# B&R Automation Studio project ACOPOSInverterTool
Automation Studio 4.12.3.127 SP; technology packages: mapp 5.23.0, mappFramework 1.0.0, mappMotion 5.23.0, mappView 5.23.0

## Configuration Config1

CPU 4PPC70.0573-20B, AutomationRuntime E4.93, Build 4.1.2, Safety 0.0, Vc V4.72.5

### Task classes (Cpu.sw)
```
Cyclic#4:
  Main <- Main.prg
NcDataObjects: mcdrivelog
Binaries: TCLang, arsvcreg, FWRules, mvLoader, TCData, udbdef, arflatprv, arcoal, iomap, asfw, Role, ashwd, Config, Config_1, TC, arconfig, sysconf, User, ashwac
Libraries: AsEPL, runtime, MpServer, MpAlarmX, MpBase, astime, MpRecipe, sys_lib, MpCom, AsIecCon, AsMath, asstring, FileIO, AsXml, standard, ArEventLog, McBase, arssl, SfDomVis, MpSfDomMgr, dataobj, asiodiag, SfDomDrv, aruser, asusb, AsTCP, MpAxis, McAxis, McAcpAx, AsIORTI
```

### Hardware
```
4PPC70_0573_20B : 4PPC70.0573-20B v1.5.4.0
  Connector IF2:
    ActivateDevice = 1
    Mode = Manual
    InternetAddress = 192.168.0.20
    SubnetMask = 255.255.255.0
    InaPort = 11160
    ActivateSnmp = 2
    ActivateModbus = 1
    NumSlaves = -1
    NumAllBlocks = -1
    MemSizeIn = -1
    MemSizeOut = -1
    ModbusSlaveGrey = 1
  ConfigurationID = ACOPOSInverterTool_Config1
  Simulation = 1
  XLinkUseDefault = 0
  XLinkDuration = 2000
  Cyclic1Duration = 2000
  Cyclic1Tolerance = 0
  FileDevice1
  FileDeviceName1 = USER
  FileDevicePath1 = USER_PATH
  ActivateOpcUa = 1
  OpcUaInformationModels_PV_Version = 1
  KeyMappingFile = VC\4PPC70_0573_20B.dis
8I66xxxxxxx.0P-xxx : 8I66xxxxxxx.0P-xxx v2.5.1.0  [PLK1 -> 4PPC70_0573_20B.IF1 (NodeNumber=2) [Cable Type=PowerlinkCable, Length=10, Version=1.0.0.3]]
  Supervision = off
  FunctionModel = Standard
  UnitOfSetpoint = Rpm
  IOM_AIDP1 = RFR_D
  IOM_AIDP2 = FRO_D
  IOM_AIDP3 = OTRN
  IOM_AIDP4 = UOP
  IOM_AIDP5 = LCR
  IOM_AIDP6 = SLCR
  IOM_AIDP7 = OPR
  IOM_AIDP8 = ULN
  IOM_AIDP9 = THR
  IOM_AIDP10 = THD
  FunctionModel_ACPi = Template50_SYN
  Sel_NameplateMask = 8Ix6T200037_IEC
  Sel_TUN = MANU
  Sel_References = Hz
  Cfg_FLR = 1
```

### IoMap.iom - 4PPC70_0573_20B/IoMap.iom
```iecst
VAR_CONFIG
	::Main:controlWord AT %QW."8I66xxxxxxx.0P-xxx".CMDD_Output;
	::Main:errorWord AT %IW."8I66xxxxxxx.0P-xxx".ERRD_Input;
	::Main:statusWord AT %IW."8I66xxxxxxx.0P-xxx".ETAD_Input;
	::Main:hmiCom.cmd.Speed AT %QW."8I66xxxxxxx.0P-xxx".LFRD_Output;
	::Main:hmiCom.cmd.ActualSpeed  AT %IW."8I66xxxxxxx.0P-xxx".RFRD_Input;
	::Main:hmiCom.cmd.Freq AT %IW."8I66xxxxxxx.0P-xxx".FRO_Input;
	::Main:hmiCom.cmd.ActualFreq AT %IW."8I66xxxxxxx.0P-xxx".RFR_Input;
END_VAR
```

## Logical view

Binary libraries used (declarations not repeated): operator, runtime, astime, AsIecCon, AsEPL, sys_lib, AsMath, asstring, FileIO, AsXml, standard, ArEventLog, AsTCP, McBase, MpAxis, McAcpAx, McAxis, MpBase, MpRecipe, MpAlarmX, MpCom 5.23.0, MpServer, AsIORTI


### Program Logical/Main (IEC)

#### Main.st - Init, cyclic, exit code
```iecst
//
PROGRAM _INIT
//
//	(*Enable FB Blocks*) // ???
//	eplWriteBlock.enable 	:= TRUE;
//	eplReadBlock.enable 	:= TRUE;
//
END_PROGRAM
//
PROGRAM _CYCLIC
//
//	//Mappview String Handling Task
	stringhandling;
//
//	//By Default Remove Ability to Control Axis
//	//controlEnable := FALSE;
//
//	//Assign pDevice
//
//	IF hmiCom.PowerLinkPathDefault THEN
//		//If a null pointer is specified, the function block uses the first POWERLINK interface
//		eplReadBlock.pDevice 	:= 0;
//		eplWriteBlock.pDevice 	:= 0;
//	ELSIF NOT hmiCom.PowerLinkPathDefault THEN
//
//		pDevice :=
//		eplReadBlock.pDevice 	:= ADR(pDevice);
//		eplWriteBlock.pDevice 	:= ADR(pDevice);
	//Assign NodeNumber from Vis
	eplReadBlock.node		:= hmiCom.NodeNumber;
	eplWriteBlock.node		:= hmiCom.NodeNumber;
//
//
	CASE state OF

		WAIT:

			//Run Startup Routine
			IF startupRoutine AND hmiCom.NodeNumber <> 0 THEN
				startup;
			END_IF

			//Run Main Routine
			IF startupDone THEN
				j := 0;
				i := 0;
				startupRoutine := FALSE;
				state := RUN;
			END_IF

		RUN:

			CASE runstate OF

				WAITING:

					hmiCom.Reading := FALSE;
					hmiCom.Writing := FALSE;

					IF hmiCom.cmd.loadParams = 1 THEN
						hmiCom.status.readInpr := TRUE;
						hmiCom.status.ReadDone := FALSE;
						runstate := READING;
					END_IF

					IF hmiCom.cmd.saveParams = 1 THEN
						hmiCom.status.writeInpr := TRUE;
						hmiCom.status.WriteDone := FALSE;
						runstate := WRITING;
					END_IF

				READING:
					hmiCom.Reading := TRUE;
					CASE readstate OF
						READPARAMS:
							IF readBools[i] THEN 		// readBools[i] should all be 1. Added for future use
								eplReadBlock.enable			:= TRUE;
								eplReadBlock.index 			:= eplReadBuffer[i].index;
								eplReadBlock.subindex 		:= eplReadBuffer[i].subindex;
								eplReadBlock.datalen 		:= 2;	//2 bytes
								eplReadBlock.pData 		:= eplReadBuffer[i].pData;
								eplReadBuffer[i].status 	:= eplReadBlock.status;
								eplReadBuffer[i].errorinfo	:= eplReadBlock.errorinfo;
							END_IF

							//Check For Error, then move to iterate counter
							IF eplReadBlock.status = 0 THEN
								readstate 					:= ITERATEREADCOUNT;
							ELSIF NOT (eplReadBlock.status = 0 OR eplReadBlock.status = 65535 OR eplReadBlock.status = 65534) THEN
								readstate := READERROR;
								state := GLOBALERROR;
							END_IF

						ITERATEREADCOUNT:

							//Turn off enable
							eplReadBlock.enable	:= FALSE;

							//Iterate Counter
							IF i = MAXINDEX THEN
//								hmiCom.status.readInpr := FALSE;
//								hmiCom.status.ReadDone := TRUE;
								i := 0;
								readstate := READPARAMS;
								runstate := WAITING;
								hmiCom.status.readInpr := FALSE;
								hmiCom.status.ReadDone := TRUE;
							ELSE
								i := i + 1;
							END_IF
							//Send Back to Reading State
							readstate 	:= READPARAMS;

						READERROR:

							IF hmiCom.cmd.Reset = TRUE THEN

							END_IF

					END_CASE

				WRITING:
					hmiCom.Writing := FALSE;
					CASE writestate OF

						WRITEPARAMS:

							IF writeBools[j] THEN
								eplWriteBlock.index				:= eplReadBuffer[j].index;
								eplWriteBlock.subindex			:= eplReadBuffer[j].subindex;
								eplWriteBlock.datalen 			:= SIZEOF(readData.ADC);	//Any will do since the max is 2 bytes
								eplWriteBlock.pData 			:= eplReadBuffer[i].pData;
								eplWriteBuffer[j].status 		:= eplWriteBlock.status;
								eplWriteBuffer[j].errorinfo		:= eplWriteBlock.errorinfo;

								eplReadBlock.enable			:= TRUE;
							END_IF

							IF eplWriteBlock.status = 65535 THEN
								writestate 					:= ITERATEWRITECOUNT;
							END_IF

						ITERATEWRITECOUNT:
							//Turn off enable
							eplWriteBlock.enable	:= FALSE;

							//Iterate Counter
							IF j = MAXINDEX THEN
								j := 0;
								hmiCom.status.writeInpr := FALSE;
								hmiCom.status.WriteDone := TRUE;
								writestate := WRITEPARAMS;
								runstate := WAITING;
							ELSE
								j := j + 1;
							END_IF

							//Send Back to writing state
							writestate 	:= WRITEPARAMS;

						WRITEERROR:

					END_CASE

			END_CASE

		GLOBALERROR:

	END_CASE
//
//
//
	eplWriteBlock();

IF startupDone THEN
	eplReadBlock();
END_IF

END_PROGRAM
//
PROGRAM _EXIT
//	(* Insert code here *)
//
END_PROGRAM
//
```

#### Types.typ - Local data types
```iecst
(**********************************HMI VARIABLES***********************************************************)

TYPE
	hmiCommTyp : 	STRUCT  (*HMI communication structure*)
		ReadWriteBuffer : DataBufferTyp; (*Command to write*)
		InverterModel : invertermodel_enum;
		InverterModelInt : USINT;
		InverterModelString : STRING[20];
		MotorType : motortype_enum;
		PowerLinkPathDefault : BOOL; (*Set to true if there's only 1 powerlink interface on the PC*)
		PowerLinkPath : powerlinkPathTyp;
		NodeNumber : USINT; (*Node number of ACOPOS Inverter*)
		Params : paramsTyp; (*Data used in ParamsContent*)
		cmd : hmiCmdTyp;
		status : hmiStatusTyp;
		unitMonitoring : unitMonitoringTyp;
		Writing : BOOL;
		Reading : BOOL;
		selectedNRDIndex : USINT;
		selectedSFTValue : STRING[3];
		selectedSTFInt : USINT;
		selectedCFTValue : STRING[3];
		selectedCFTInt : USINT;
		selectedCTTValue : STRING[3];
		selectedCTTint : USINT;
		selectedAstValue : STRING[3];
		selectedInverter : STRING[80];
		selectedInverterINT : USINT;
		selectedMotorType : STRING[3];
		selectedMotorINT : USINT;
	END_STRUCT;
	invertermodel_enum :
		( (*ACOPOS Inverter Model enumeration*)
		P66 := 66,
		P76 := 76,
		P86 := 86
		);
	motortype_enum :
		(
		Asynchronous := 0,
		Synchronous := 1
		);
	powerlinkPathTyp : 	STRUCT  (*Carries path strings to build "SL<x>.SS<y>.IF<Z>"*)
		SLnumber : STRING[8]; (*SLx*)
		SSnumber : STRING[8]; (*SSy*)
		IFnumber : STRING[8]; (*IFz*)
	END_STRUCT;
	hmiCmdTyp : 	STRUCT
		Speed : INT;
		ActualSpeed : INT;
		Freq : INT;
		ActualFreq : INT;
		CMDD : UINT;
		loadParams : BOOL;
		saveParams : BOOL;
		Reset : BOOL;
	END_STRUCT;
	hmiStatusTyp : 	STRUCT
		ERRD : STRING[20];
		ETAD : STRING[20];
		FirmwareVersion : STRING[20];
		readInpr : BOOL;
		writeInpr : BOOL;
		ReadDone : USINT;
		WriteDone : USINT;
	END_STRUCT;
END_TYPE

(**********************************State Enumerations*********************************************************)

TYPE
	state_enum :
		(
		WAIT,
		RUN,
		GLOBALERROR
		);
	runstate_enum :
		(
		WAITING,
		READING,
		WRITING
		);
	startupstate_enum :
		(
		INITIALIZE,
		COPY,
		FIRSTREAD,
		DONE
		);
	readstate_enum :
		(
		READPARAMS,
		ITERATEREADCOUNT,
		READERROR
		);
	writestate_enum :
		(
		WRITEPARAMS,
		ITERATEWRITECOUNT,
		WRITEERROR,
		ALGR (*Status word of user defined alarm groups*)
		);
END_TYPE

(**********************************Parameter Structures******************************************************)

TYPE
	eplParTyp : 	STRUCT
		index : UINT; (*Number of the index entry to be written.
*)
		subindex : USINT; (*Number of the subindex entry to be written.
*)
		pData : UDINT; (*Pointer to the data to be written. This data must remain constant as long as the function block returns ERR_BUSY.
*)
		datalen : UDINT; (*Length of the data to be written.
*)
		status : UINT; (*Error number (0 = no error).
*)
		errorinfo : UDINT; (*SDO Abort Code (if status = ERR_ASEPL_ACCESS_FAILED)
*)
		name : STRING[50]; (*Name of Parameter*)
		measurementUnit : measurementunit_enum; (*Unit of measurement for the data*)
		conversionFactor : REAL; (*Conversion factor from data to measurement unit*)
	END_STRUCT;
	DataBufferTyp : 	STRUCT
		NSP : UINT;
		FRS : UINT;
		UNS : UINT;
		NCR : UINT;
		COSINE : UINT;
		NPR : UINT;
		TUN : WORD; (*0 - no action, 1- tune, 2 - delete tuning*)
		RSA : UINT;
		LFA : UINT;
		IDA : UINT;
		TRA : UINT;
		SFR : UINT;
		SFT : WORD; (*Heat Optimized (1), Noise Optimized (2)*)
		NRD : USINT; (*Vary PWM period for Noise reduction- No (0), Yes (1)*)
		CTT : WORD; (*(UUC)/Sensorless Flux Vector 	(0)
							 (STD)/Standard 			  	(3)
							 (UF5)/ (V/F 5pts) 				(4)
							 (SYN)/ Synchronous motor		(5)
							 (UFQ)/ (V/F QUAD.) 			(6)
							 (NLD)/Energy Saving			(7)*)
		SPGU : UINT; (*For Standard mode: *)
		SPG : UINT; (*For Vector control:*)
		FFH : UINT;
		CRTF : UINT;
		SLP : UINT;
		UFR : UINT;
		BOA : WORD; (*Boost Enum, 0 Boost inactive, 1 boost dynamic, 2 boost static*)
		FAB : UINT;
		BOO : INT;
		PFL : UINT;
		F1 : UINT;
		U1 : UINT;
		F2 : UINT;
		U2 : UINT;
		F3 : UINT;
		U3 : UINT;
		F4 : UINT;
		U4 : UINT;
		F5 : UINT;
		U5 : UINT;
		SIT : UINT;
		SFC : UINT;
		JFH : UINT;
		JPF : UINT;
		JF2 : UINT;
		JF3 : UINT;
		SPA : UINT;
		SPAT : UINT;
		SPD : UINT;
		SPDT : UINT;
		RPT : WORD; (*Enum - Linear Ramp (0), S-ramp (1), U-Ramp (2), Customized (3)*)
		ADC : WORD; (*Enum - No DC inject(0), Yes (1), Continuous DC inj brake (2)*)
		FLR : WORD; (*Enum - catch spinning loads No(0), yes(1)*)
		SDC1 : UINT;
		TDC1 : UINT;
		SDC2 : UINT;
		TDC2 : UINT;
		BRA : WORD; (*Enum - Braking cmd transistor(No) (0), Dec ramp adapt assinged (YES) (1), Dynamic high torque (2)*)
		DCF : UINT;
		IDC : UINT;
		TDI : USINT;
		IDC2 : UINT;
		TDC : UINT;
		ULT : UINT;
		LUL : UINT;
		RMUD : UINT;
		LUN : UINT;
		FTU : UINT;
		TOL : UINT;
		LOC : UINT;
		FTO : UINT;
		ITH : UINT;
		I2TA : UINT; (*Enumeration - 0 (no), 1 (yes)*)
		OTR : USINT; (*Monitored Value for Torque*)
		MAINS : UINT;
		PPNS : UINT; (*Synchronous Motor Pole Pair*)
		NSPS : UINT; (*Sync motor speed*)
		NCRS : UINT; (*Sync motor current*)
		TQS : UINT; (*Sync motor torque*)
		RSAS : UINT; (*Stator resistance (Sync)*)
		LDS : UINT; (*Direct inductance (Sync)*)
		LQS : UINT; (*Quadrature Inductance (Sync)*)
		PHS : UINT; (*Sync EMF (Voltage) constant*)
		AST : UINT; (*Synchronous Motor Construction Type*)
	END_STRUCT;
	paramsTyp : 	STRUCT
		UnitMonitoring : unitMonitoringTyp; (*Datapoints used in Units/Monitoring tab*)
	END_STRUCT;
	unitMonitoringTyp : 	STRUCT
		MeasurementUnit : measurementunit_enum;
		Units : ARRAY[0..7]OF unitTyp;
	END_STRUCT;
	unitTyp : 	STRUCT
		Unit : unit_enum; (*Unit being monitored*)
		String : STRING[80]; (*String of Description*)
		PowerlinkIndex : UINT; (*Powerlink Index*)
		PowerlinkSubindex : UINT; (*Powerlink Subindex*)
	END_STRUCT;
	measurementunit_enum :
		(
		Undefined := 0,
		Hz := 1, (*Hertz*)
		RPM := 2, (*RPM*)
		Volts := 3, (*Volts*)
		Amps := 4, (*Amperes*)
		Percent := 5, (*%*)
		NewtonMeter := 6, (*Newton-Meter*)
		Seconds := 7, (*Seconds*)
		Ohm := 8, (*Ohm*)
		Millihenry := 9 (*mH*)
		);
	unit_enum :
		( (*Enumeration containing the units that can be monitored on the inverter*)
		UNDEFINED, (*undefined*)
		HMIS, (*Device specific error code*)
		ETI, (*Internal status word*)
		THR, (*Thermal status of motor (i^2 * t)*)
		THD, (*Thermal status of drive [%]*)
		I2TM, (*Overcurrent status of motor (I^2 * t)[%]*)
		PTCI, (*Status word of PTC on DI6*)
		ALGROUP, (*Status word of user defined alarm groups*)
		STOS, (*Status word of STO (safe torque off)*)
		SS1S, (*Status word of SS1 (safe speed 1)*)
		SLSS, (*Status word of SLS (safely limit speed)*)
		SMSS, (*Status word of SMS (safe maximum speed)*)
		GDLS, (*Status word of GDL (guard door locking)*)
		ETAD, (*Status word (as BOOL)*)
		RFR, (*Frequency value [Hz] (PWM output)*)
		SRFR, (*unfiltered raw value of RFR [Hz]*)
		FRO, (*Frequency reference after a ramp [Hz] (value for PWM control)*)
		FRH, (*Frequency reference after n limitation [Hz] (value before ramp)*)
		FRHD, (*Speed reference after n limitation [rpm]*)
		OTR, (*Torque [%] (according to DS402)*)
		SOTR, (*unfiltered incremental value of OTR*)
		OTRN, (*Torque [Nm]*)
		UOP, (*Voltage [V] (PWM output) *)
		LCR, (*Current [A] (PWM output)*)
		SLCR, (*unfiltered raw value of LCR [A]*)
		OPR, (*Power [%] (PWM output)*)
		SOPR, (*unfiltered raw value of OPR [%]*)
		ULN, (*Mains voltage level [V]*)
		SULN, (*unfiltered raw valueof ULN [V]*)
		AI1R, (*Status word of analog input 1*)
		AI1RUINT, (*Status word (as UINT)*)
		AI2R, (*Status word of analog input 2*)
		AI2RUINT, (*Status word (as UINT)*)
		AI3R, (*Status word of analog input 3*)
		AI3RUINT, (*Status word (as UINT)*)
		IL1R, (*Status word of digital inputs*)
		IL1RBOOL, (*Status word (as BOOL)*)
		HSC, (*Edge counter on DI5*)
		PIFR, (*Pulse input on DI5 [0 .. 8192]*)
		PFRC, (*Pulse input on DI5 [Hz] *)
		FQS, (*Frequency meter on DI5 [Hz] (processed value)*)
		AO1I, (*Status word of analog output 1*)
		OL1I, (*Status word of digital outputs*)
		OL1IBOOL, (*Status word (as BOOL)*)
		NCRS (*Set to NCR(S) (motor nominal current)*)
		);
	ast_change_enum :
		(
		NOCHANGE,
		VISCHANGE,
		DRIVECHANGE
		);
END_TYPE

(***********************************Parameter enumerations************************************************)
```

#### Variables.var - Local variables
```iecst
(*************************************EPL Stuff************************************************************************)
VAR
	eplWriteBlock : EplSDOWrite; (*This function block is used to write a node's object entries when using an SDO transfer that is constantly running in the background.
*)
	eplReadBlock : EplSDORead; (*This function block is used to read a node's object entries when using an SDO transfer that is constantly running in the background.
*)
	eplReadBuffer : ARRAY[0..MAXINDEX] OF eplParTyp; (*Array of Inputs for the Read FB*)
	eplWriteBuffer : ARRAY[0..MAXINDEX] OF eplParTyp; (*Array of Inputs for the Write FB (Open to see parameters)*)
	readBools : ARRAY[0..MAXINDEX] OF BOOL;
	writeBools : ARRAY[0..MAXINDEX] OF BOOL;
	readData : DataBufferTyp;
	writeData : DataBufferTyp;
	pDevice : STRING[80]; (*Device name of the POWERLINK interface (syntax: SL<x>.SS<y>.IF<z>). If a null pointer is specified, the function block uses the first POWERLINK interface on the system.
*)
	state : state_enum; (*State enumeration variable*)
	runstate : runstate_enum;
	readstate : readstate_enum; (*State enumeration variable*)
	writestate : writestate_enum; (*State enumeration variable*)
	startupstate : startupstate_enum;
	aststate : ast_change_enum;
	i : USINT; (*for loop variable*)
	j : USINT; (*loop variable 2*)
	k : USINT; (*loop variable 3*)
END_VAR
VAR CONSTANT
	MAXINDEX : USINT := 77; (*Maximum index*)
END_VAR
VAR
	hmiCom : hmiCommTyp;
	addressBook : USINT;
	startupRoutine : BOOL;
	startupDone : BOOL;
	oldAstVis : STRING[3];
	oldAstDrive : UINT;
END_VAR
(**************************************Test Stuff***********************************************************************)
VAR
	controlWord : UINT; (*CMDD*)
	errorWord : UINT; (*ERRD*)
	statusWord : UINT; (*ETAD*)
	setpointRead : INT; (*FROD*)
	setpointWrite : INT; (*LFRD*)
	feedbackValue : INT; (*RFRD*)
	controlEnable : BOOL; (*Boolean to prevent writing to EPL while controlling the axis*)
	firmwareVersion : UDINT;
	hardwareVariant : UDINT;
END_VAR
(*************************************Hmi Comm Stuff********************************************************************)
VAR
	comm : hmiCommTyp;
END_VAR
```

#### stringhandling.st
```iecst
ACTION stringhandling:

		//Inverter Model

		//Motor Type

		hmiCom.selectedMotorINT := STRING_TO_USINT(hmiCom.selectedMotorType);

		//Monitored Units

		FOR k := 0  TO 7 DO
			CASE hmiCom.Params.UnitMonitoring.Units[i].Unit OF

			UNDEFINED:
				hmiCom.Params.UnitMonitoring.Units[k].String 			:= 'Undefined';
				hmiCom.Params.UnitMonitoring.Units[k].PowerlinkIndex 	:= 16#0;
				hmiCom.Params.UnitMonitoring.Units[k].PowerlinkSubindex := 16#0;
				hmiCom.Params.UnitMonitoring.MeasurementUnit 			:= Undefined;
			HMIS:
				//A bunch of different HMIS in the sheet, using the first
				hmiCom.Params.UnitMonitoring.Units[k].String 			:= 'Device specific error code';
				hmiCom.Params.UnitMonitoring.Units[k].PowerlinkIndex 	:= 16#202B;
				hmiCom.Params.UnitMonitoring.Units[k].PowerlinkSubindex := 16#16;
				hmiCom.Params.UnitMonitoring.MeasurementUnit 			:= Undefined;
			ETI:
				//A bunch of different ETI in the sheet, using the first
				hmiCom.Params.UnitMonitoring.Units[k].String 			:= 'Internal status word';
				hmiCom.Params.UnitMonitoring.Units[k].PowerlinkIndex 	:= 16#202A;
				hmiCom.Params.UnitMonitoring.Units[k].PowerlinkSubindex := 16#15;
				hmiCom.Params.UnitMonitoring.MeasurementUnit 			:= Undefined;
			THR:
				hmiCom.Params.UnitMonitoring.Units[k].String 			:= 'Thermal status of motor (i^2 * t)';
				hmiCom.Params.UnitMonitoring.Units[k].PowerlinkIndex 	:= 16#2042;
				hmiCom.Params.UnitMonitoring.Units[k].PowerlinkSubindex := 16#1F;
				hmiCom.Params.UnitMonitoring.MeasurementUnit 			:= Undefined;
			THD:
				hmiCom.Params.UnitMonitoring.Units[k].String 			:= 'Thermal status of drive [%]';
				hmiCom.Params.UnitMonitoring.Units[k].PowerlinkIndex 	:= 16#2002;
				hmiCom.Params.UnitMonitoring.Units[k].PowerlinkSubindex := 16#0A;
				hmiCom.Params.UnitMonitoring.MeasurementUnit 			:= Undefined;
			I2TM:
				hmiCom.Params.UnitMonitoring.Units[k].String 			:= 'Overcurrent status of motor (I^2 * t)[%]';
				hmiCom.Params.UnitMonitoring.Units[k].PowerlinkIndex 	:= 16#2042;
				hmiCom.Params.UnitMonitoring.Units[k].PowerlinkSubindex := 16#23;
				hmiCom.Params.UnitMonitoring.MeasurementUnit 			:= Undefined;
			PTCI:
				hmiCom.Params.UnitMonitoring.Units[k].String 			:= 'Status word of PTC on DI6';
				hmiCom.Params.UnitMonitoring.Units[k].PowerlinkIndex 	:= 16#2066;
				hmiCom.Params.UnitMonitoring.Units[k].PowerlinkSubindex := 16#04;
				hmiCom.Params.UnitMonitoring.MeasurementUnit 			:= Undefined;
			ALGROUP:
				//Not sure this exists on the drive, link through IO mapping
				hmiCom.Params.UnitMonitoring.Units[k].String 			:= 'Status word of user defined alarm groups';
				hmiCom.Params.UnitMonitoring.Units[k].PowerlinkIndex 	:= 16#0;
				hmiCom.Params.UnitMonitoring.Units[k].PowerlinkSubindex := 16#0;
				hmiCom.Params.UnitMonitoring.MeasurementUnit 			:= Undefined;
			STOS:
				hmiCom.Params.UnitMonitoring.Units[k].String 			:= 'Status word of STO (safe torque off)';
				hmiCom.Params.UnitMonitoring.Units[k].PowerlinkIndex 	:= 16#0;
				hmiCom.Params.UnitMonitoring.Units[k].PowerlinkSubindex := 16#0;
				hmiCom.Params.UnitMonitoring.MeasurementUnit 			:= Undefined;
			SS1S:
				hmiCom.Params.UnitMonitoring.Units[k].String 			:= 'Status word of SS1 (safe speed 1)';
				hmiCom.Params.UnitMonitoring.Units[k].PowerlinkIndex 	:= 16#207B;
				hmiCom.Params.UnitMonitoring.Units[k].PowerlinkSubindex := 16#10;
				hmiCom.Params.UnitMonitoring.MeasurementUnit 			:= Undefined;
			SLSS:
				hmiCom.Params.UnitMonitoring.Units[k].String 			:= 'Status word of SLS (safely limit speed)';
				hmiCom.Params.UnitMonitoring.Units[k].PowerlinkIndex 	:= 16#207B;
				hmiCom.Params.UnitMonitoring.Units[k].PowerlinkSubindex := 16#05;
				hmiCom.Params.UnitMonitoring.MeasurementUnit 			:= Undefined;
			SMSS:
				hmiCom.Params.UnitMonitoring.Units[k].String 			:= 'Status word of SMS (safe maximum speed)';
				hmiCom.Params.UnitMonitoring.Units[k].PowerlinkIndex 	:= 16#207B;
				hmiCom.Params.UnitMonitoring.Units[k].PowerlinkSubindex := 16#055;
				hmiCom.Params.UnitMonitoring.MeasurementUnit 			:= Undefined;
			GDLS:
				hmiCom.Params.UnitMonitoring.Units[k].String 			:= 'Status word of GDL (guard door locking)';
				hmiCom.Params.UnitMonitoring.Units[k].PowerlinkIndex 	:= 16#207B;
				hmiCom.Params.UnitMonitoring.Units[k].PowerlinkSubindex := 16#05E;
				hmiCom.Params.UnitMonitoring.MeasurementUnit 			:= Undefined;
			ETAD:
				hmiCom.Params.UnitMonitoring.Units[k].String 			:= 'Drive Status Word';
				hmiCom.Params.UnitMonitoring.Units[k].PowerlinkIndex 	:= 16#2038;
				hmiCom.Params.UnitMonitoring.Units[k].PowerlinkSubindex := 16#04;
				hmiCom.Params.UnitMonitoring.MeasurementUnit 			:= Undefined;
			RFR:
				hmiCom.Params.UnitMonitoring.Units[k].String 			:= 'Frequency value [Hz] (PWM output)';
				hmiCom.Params.UnitMonitoring.Units[k].PowerlinkIndex 	:= 16#2002;
				hmiCom.Params.UnitMonitoring.Units[k].PowerlinkSubindex := 16#03;
				hmiCom.Params.UnitMonitoring.MeasurementUnit 			:= Hz;
			SRFR:
				hmiCom.Params.UnitMonitoring.Units[k].String 			:= 'Unfiltered raw value of RFR [Hz]';
				hmiCom.Params.UnitMonitoring.Units[k].PowerlinkIndex 	:= 16#2038;
				hmiCom.Params.UnitMonitoring.Units[k].PowerlinkSubindex := 16#04;
				hmiCom.Params.UnitMonitoring.MeasurementUnit 			:= Hz;
			FRO:
				hmiCom.Params.UnitMonitoring.Units[k].String 			:= 'Frequency reference after a ramp [Hz] (value for PWM control)';
				hmiCom.Params.UnitMonitoring.Units[k].PowerlinkIndex 	:= 16#203C;
				hmiCom.Params.UnitMonitoring.Units[k].PowerlinkSubindex := 16#16;
				hmiCom.Params.UnitMonitoring.MeasurementUnit 			:= Hz;
			FRH:
				hmiCom.Params.UnitMonitoring.Units[k].String 			:= 'Frequency reference after n limitation [Hz] (value before ramp)';
				hmiCom.Params.UnitMonitoring.Units[k].PowerlinkIndex 	:= 16#203C;
				hmiCom.Params.UnitMonitoring.Units[k].PowerlinkSubindex := 16#16;
				hmiCom.Params.UnitMonitoring.MeasurementUnit 			:= Hz;
			FRHD:
				hmiCom.Params.UnitMonitoring.Units[k].String 			:= 'Speed reference after n limitation [rpm]';
				hmiCom.Params.UnitMonitoring.Units[k].PowerlinkIndex 	:= 16#2039;
				hmiCom.Params.UnitMonitoring.Units[k].PowerlinkSubindex := 16#06;
				hmiCom.Params.UnitMonitoring.MeasurementUnit 			:= RPM;
			OTR:
				hmiCom.Params.UnitMonitoring.Units[k].String 			:= 'Torque [%] (according to DS402)';
				hmiCom.Params.UnitMonitoring.Units[k].PowerlinkIndex 	:= 16#2002;
				hmiCom.Params.UnitMonitoring.Units[k].PowerlinkSubindex := 16#06;
				hmiCom.Params.UnitMonitoring.MeasurementUnit 			:= Percent;
			SOTR:
				hmiCom.Params.UnitMonitoring.Units[k].String 			:= 'Unfiltered incremental value of OTR';
				hmiCom.Params.UnitMonitoring.Units[k].PowerlinkIndex 	:= 16#2002;
				hmiCom.Params.UnitMonitoring.Units[k].PowerlinkSubindex := 16#1B;
				hmiCom.Params.UnitMonitoring.MeasurementUnit 			:= Percent;
			OTRN:
				//Doesn't exist on drive, link through IO mapping
				hmiCom.Params.UnitMonitoring.Units[k].String 			:= 'Torque in Newton-meters';
				hmiCom.Params.UnitMonitoring.Units[k].PowerlinkIndex 	:= 16#0;
				hmiCom.Params.UnitMonitoring.Units[k].PowerlinkSubindex := 16#0;
				hmiCom.Params.UnitMonitoring.MeasurementUnit 			:= NewtonMeter;
			UOP:
				hmiCom.Params.UnitMonitoring.Units[k].String 			:= 'Voltage [V] (PWM output)';
				hmiCom.Params.UnitMonitoring.Units[k].PowerlinkIndex 	:= 16#2002;
				hmiCom.Params.UnitMonitoring.Units[k].PowerlinkSubindex := 16#09;
				hmiCom.Params.UnitMonitoring.MeasurementUnit 			:= Volts;
			LCR:
				hmiCom.Params.UnitMonitoring.Units[k].String 			:= 'Current [A] (PWM output)';
				hmiCom.Params.UnitMonitoring.Units[k].PowerlinkIndex 	:= 16#2002;
				hmiCom.Params.UnitMonitoring.Units[k].PowerlinkSubindex := 16#05;
				hmiCom.Params.UnitMonitoring.MeasurementUnit 			:= Amps;
			SLCR:
				hmiCom.Params.UnitMonitoring.Units[k].String 			:= 'Unfiltered raw value of LCR [A]';
				hmiCom.Params.UnitMonitoring.Units[k].PowerlinkIndex 	:= 16#2002;
				hmiCom.Params.UnitMonitoring.Units[k].PowerlinkSubindex := 16#19;
				hmiCom.Params.UnitMonitoring.MeasurementUnit 			:= Amps;
			OPR:
				hmiCom.Params.UnitMonitoring.Units[k].String 			:= 'Power [%] (PWM output)';
				hmiCom.Params.UnitMonitoring.Units[k].PowerlinkIndex 	:= 16#2002;
				hmiCom.Params.UnitMonitoring.Units[k].PowerlinkSubindex := 16#0C;
				hmiCom.Params.UnitMonitoring.MeasurementUnit 			:= Percent;
			SOPR:
				hmiCom.Params.UnitMonitoring.Units[k].String 			:= 'unfiltered raw value of OPR [%]';
				hmiCom.Params.UnitMonitoring.Units[k].PowerlinkIndex 	:= 16#2002;
				hmiCom.Params.UnitMonitoring.Units[k].PowerlinkSubindex := 16#5B;
				hmiCom.Params.UnitMonitoring.MeasurementUnit 			:= Percent;
			ULN:
				hmiCom.Params.UnitMonitoring.Units[k].String 			:= 'Mains voltage level [V]';
				hmiCom.Params.UnitMonitoring.Units[k].PowerlinkIndex 	:= 16#2002;
				hmiCom.Params.UnitMonitoring.Units[k].PowerlinkSubindex := 16#08;
				hmiCom.Params.UnitMonitoring.MeasurementUnit 			:= Volts;
			SULN:
				hmiCom.Params.UnitMonitoring.Units[k].String 			:= 'Unfiltered raw valueof ULN [V]';
				hmiCom.Params.UnitMonitoring.Units[k].PowerlinkIndex 	:= 16#2002;
				hmiCom.Params.UnitMonitoring.Units[k].PowerlinkSubindex := 16#1E;
				hmiCom.Params.UnitMonitoring.MeasurementUnit 			:= Volts;
			AI1R:
				hmiCom.Params.UnitMonitoring.Units[k].String 			:= 'Analog Input 1';
				hmiCom.Params.UnitMonitoring.Units[k].PowerlinkIndex 	:= 16#2016;
				hmiCom.Params.UnitMonitoring.Units[k].PowerlinkSubindex := 16#21;
				hmiCom.Params.UnitMonitoring.MeasurementUnit 			:= Undefined;
			AI2R:
				hmiCom.Params.UnitMonitoring.Units[k].String 			:= 'Analog Input 2';
				hmiCom.Params.UnitMonitoring.Units[k].PowerlinkIndex 	:= 16#2016;
				hmiCom.Params.UnitMonitoring.Units[k].PowerlinkSubindex := 16#22;
				hmiCom.Params.UnitMonitoring.MeasurementUnit 			:= Undefined;
			AI3R:
				hmiCom.Params.UnitMonitoring.Units[k].String 			:= 'Analog Input 3';
				hmiCom.Params.UnitMonitoring.Units[k].PowerlinkIndex 	:= 16#2016;
				hmiCom.Params.UnitMonitoring.Units[k].PowerlinkSubindex := 16#23;
				hmiCom.Params.UnitMonitoring.MeasurementUnit 			:= Undefined;
			IL1R:
				hmiCom.Params.UnitMonitoring.Units[k].String 			:= 'Status word of digital inputs';
				hmiCom.Params.UnitMonitoring.Units[k].PowerlinkIndex 	:= 16#2016;
				hmiCom.Params.UnitMonitoring.Units[k].PowerlinkSubindex := 16#03;
				hmiCom.Params.UnitMonitoring.MeasurementUnit 			:= Undefined;
			HSC:
				hmiCom.Params.UnitMonitoring.Units[k].String 			:= 'Edge counter on DI5 (High Speed Counter)';
				hmiCom.Params.UnitMonitoring.Units[k].PowerlinkIndex 	:= 16#2067;
				hmiCom.Params.UnitMonitoring.Units[k].PowerlinkSubindex := 16#09;
				hmiCom.Params.UnitMonitoring.MeasurementUnit 			:= Undefined;
			PIFR:
				//Doesn't exist on Schneider Side, pull from I/O map
				hmiCom.Params.UnitMonitoring.Units[k].String 			:= 'Pulse input on DI5 [0 .. 8192]';
				hmiCom.Params.UnitMonitoring.Units[k].PowerlinkIndex 	:= 16#0;
				hmiCom.Params.UnitMonitoring.Units[k].PowerlinkSubindex := 16#0;
				hmiCom.Params.UnitMonitoring.MeasurementUnit 			:= Undefined;
			PFRC:
				//Doesn't exist on Schneider Side, pull from I/O map
				hmiCom.Params.UnitMonitoring.Units[k].String 			:= 'Pulse input on DI5 [Hz]';
				hmiCom.Params.UnitMonitoring.Units[k].PowerlinkIndex 	:= 16#0;
				hmiCom.Params.UnitMonitoring.Units[k].PowerlinkSubindex := 16#0;
				hmiCom.Params.UnitMonitoring.MeasurementUnit 			:= Undefined;
			FQS:
				//Doesn't exist on Schneider Side, pull from I/O map
				hmiCom.Params.UnitMonitoring.Units[k].String 			:= 'Frequency meter on DI5 [Hz] (processed value)';
				hmiCom.Params.UnitMonitoring.Units[k].PowerlinkIndex 	:= 16#74;
				hmiCom.Params.UnitMonitoring.Units[k].PowerlinkSubindex := 16#04;
				hmiCom.Params.UnitMonitoring.MeasurementUnit 			:= Undefined;
			AO1I:
				hmiCom.Params.UnitMonitoring.Units[k].String 			:= 'Status word of analog output 1';
				hmiCom.Params.UnitMonitoring.Units[k].PowerlinkIndex 	:= 16#2016;
				hmiCom.Params.UnitMonitoring.Units[k].PowerlinkSubindex := 16#48;
				hmiCom.Params.UnitMonitoring.MeasurementUnit 			:= Undefined;
			OL1I:
				hmiCom.Params.UnitMonitoring.Units[k].String 			:= 'Status word of digital outputs';
				hmiCom.Params.UnitMonitoring.Units[k].PowerlinkIndex 	:= 16#2016;
				hmiCom.Params.UnitMonitoring.Units[k].PowerlinkSubindex := 16#0D;
				hmiCom.Params.UnitMonitoring.MeasurementUnit 			:= Undefined;
			NCRS:
				hmiCom.Params.UnitMonitoring.Units[k].String 			:= 'Nominal sync current';
				hmiCom.Params.UnitMonitoring.Units[k].PowerlinkIndex 	:= 16#2042;
				hmiCom.Params.UnitMonitoring.Units[k].PowerlinkSubindex := 16#47;
				hmiCom.Params.UnitMonitoring.MeasurementUnit 			:= Amps;
			END_CASE
	END_FOR

	//I/O mapp Word Variables

	//Two-way bindings for data providers

CASE aststate OF
	NOCHANGE:
		IF NOT (hmiCom.selectedAstValue = oldAstVis) THEN
			aststate := VISCHANGE;
		ELSIF NOT hmiCom.ReadWriteBuffer.AST = oldAstDrive THEN
			aststate := DRIVECHANGE;
		END_IF
	oldAstVis := hmiCom.selectedAstValue;
	oldAstDrive := hmiCom.ReadWriteBuffer.AST;
	VISCHANGE:
		hmiCom.ReadWriteBuffer.AST := STRING_TO_UINT(hmiCom.selectedAstValue);
		oldAstVis := hmiCom.selectedAstValue;
		oldAstDrive := hmiCom.ReadWriteBuffer.AST;
		aststate := NOCHANGE;
	DRIVECHANGE:
		hmiCom.selectedAstValue := UINT_TO_STRING(hmiCom.ReadWriteBuffer.AST);
		oldAstVis := hmiCom.selectedAstValue;
		oldAstDrive := hmiCom.ReadWriteBuffer.AST;
		aststate := NOCHANGE;
END_CASE

END_ACTION
```

#### startup.st
```iecst
ACTION startup:

	CASE startupstate OF

		INITIALIZE:

			//Initialize values for the plk adresses, etc.
			//Asynchronous Parameters from AS config:

			eplReadBuffer[0].name  	 			:= 'NSP'; //UNSIGNED
			eplReadBuffer[0].index 	 			:= 16#2042;
			eplReadBuffer[0].subindex 			:= 16#05;
			eplReadBuffer[0].measurementUnit	:= RPM;
			eplReadBuffer[0].pData				:= ADR(readData.NSP);

			eplReadBuffer[1].name  	 			:= 'FRS'; //UNSIGNED
			eplReadBuffer[1].index 	 			:= 16#2042;
			eplReadBuffer[1].subindex 			:= 16#03;
			eplReadBuffer[1].measurementUnit	:= Hz;
			eplReadBuffer[1].pData				:= ADR(readData.FRS);

			eplReadBuffer[2].name  	 			:= 'UNS'; //UNSIGNED
			eplReadBuffer[2].index 	 			:= 16#2042;
			eplReadBuffer[2].subindex 			:= 16#02;
			eplReadBuffer[2].measurementUnit	:= Volts;
			eplReadBuffer[2].pData				:= ADR(readData.UNS);

			eplReadBuffer[3].name  	 			:= 'NCR'; //UNSIGNED
			eplReadBuffer[3].index 	 			:= 16#2042;
			eplReadBuffer[3].subindex 			:= 16#04;
			eplReadBuffer[3].measurementUnit	:= Amps;
			eplReadBuffer[3].pData				:= ADR(readData.NCR);

			eplReadBuffer[4].name  	 			:= 'COS'; //UNSIGNED
			eplReadBuffer[4].index 	 			:= 16#2042;
			eplReadBuffer[4].subindex 			:= 16#07;
			eplReadBuffer[4].measurementUnit	:= Percent;
			eplReadBuffer[4].pData				:= ADR(readData.COSINE);

			eplReadBuffer[5].name  				:= 'NPR'; //UNSIGNED
			eplReadBuffer[5].index 	 			:= 16#2042;
			eplReadBuffer[5].subindex 			:= 16#0E;
			eplReadBuffer[5].pData				:= ADR(readData.NPR);

			eplReadBuffer[6].name  	 			:= 'TUN'; //0 - no action, 1- tune, 2 - delete tuning
			eplReadBuffer[6].index 	 			:= 16#2042;
			eplReadBuffer[6].subindex 			:= 16#09;
			eplReadBuffer[6].pData				:= ADR(readData.TUN);

			eplReadBuffer[7].name  	 			:= 'RSA'; //UNSIGNED
			eplReadBuffer[7].index 	 			:= 16#2042;
			eplReadBuffer[7].subindex 			:= 16#2B;
			eplReadBuffer[7].pData				:= ADR(readData.RSA);

			eplReadBuffer[8].name  	 			:= 'LFA'; //UNSIGNED
			eplReadBuffer[8].index 	 			:= 16#2042;
			eplReadBuffer[8].subindex 			:= 16#3F;
			eplReadBuffer[8].pData				:= ADR(readData.LFA);

			eplReadBuffer[9].name  	 			:= 'IDA'; //UNSIGNED
			eplReadBuffer[9].index 	 			:= 16#2042;
			eplReadBuffer[9].subindex 			:= 16#35;
			eplReadBuffer[9].pData				:= ADR(readData.IDA);

			eplReadBuffer[10].name  	 		:= 'TRA'; //UNSIGNED
			eplReadBuffer[10].index 	 		:= 16#2042;
			eplReadBuffer[10].subindex 			:= 16#44;
			eplReadBuffer[10].pData				:= ADR(readData.TRA);

			eplReadBuffer[11].name  	 		:= 'SFR'; //UNSIGNED
			eplReadBuffer[11].index 	 		:= 16#2001;
			eplReadBuffer[11].subindex 			:= 16#03;
			eplReadBuffer[11].pData				:= ADR(readData.SFR);

			eplReadBuffer[12].name  	 		:= 'SFT'; //Enumeration - Heat Optimized (1), Noise Optimized (2)
			eplReadBuffer[12].index 	 		:= 16#2001;
			eplReadBuffer[12].subindex 			:= 16#02;
			eplReadBuffer[12].pData				:= ADR(readData.SFT);

			eplReadBuffer[13].name  	 		:= 'NRD'; //Vary PWM period for Noise reduction- No (0), Yes (1)
			eplReadBuffer[13].index 	 		:= 16#2001;
			eplReadBuffer[13].subindex 			:= 16#08;
			eplReadBuffer[13].pData				:= ADR(readData.NRD);

			(* Enumeration - (UUC)/Sensorless Flux Vector 	(0)
							 (STD)/Standard 			  	(3)
							 (UF5)/ (V/F 5pts) 				(4)
							 (SYN)/ Synchronous motor		(5)
							 (UFQ)/ (V/F QUAD.) 			(6)
							 (NLD)/Energy Saving			(7)
			*)

			eplReadBuffer[14].name  	 		:= 'CTT';  //Enum see above
			eplReadBuffer[14].index 			:= 16#2042;
			eplReadBuffer[14].subindex 			:= 16#08;
			eplReadBuffer[14].measurementUnit	:= Undefined;
			eplReadBuffer[14].pData				:= ADR(readData.CTT);

			//For STD
			eplReadBuffer[15].name  	 		:= 'SPGU'; //UNSIGNED
			eplReadBuffer[15].index 	 		:= 16#2042;
			eplReadBuffer[15].subindex 			:= 16#1E;
			eplReadBuffer[15].datalen  			:= 16;
			eplReadBuffer[15].measurementUnit	:= Undefined;
			eplReadBuffer[15].pData				:= ADR(readData.SPGU);

			//For vector control
			eplReadBuffer[16].name  	 		:= 'SPG'; //UNSIGNED
			eplReadBuffer[16].index 	 		:= 16#203D;
			eplReadBuffer[16].subindex 			:= 16#04;
			eplReadBuffer[16].pData				:= ADR(readData.SPG);

			eplReadBuffer[17].name  	 		:= 'FFH'; //UNSIGNED
			eplReadBuffer[17].index 	 		:= 16#203D;
			eplReadBuffer[17].subindex 			:= 16#10;
			eplReadBuffer[17].pData				:= ADR(readData.FFH);

			eplReadBuffer[18].name  	 		:= 'CRTF'; //UNSIGNED
			eplReadBuffer[18].index 	 		:= 16#203D;
			eplReadBuffer[18].subindex 			:= 16#11;
			eplReadBuffer[18].measurementUnit 	:= Seconds;
			eplReadBuffer[18].pData				:= ADR(readData.CRTF);

			eplReadBuffer[19].name  	 		:= 'SLP'; //UNSIGNED
			eplReadBuffer[19].index 	 		:= 16#2042;
			eplReadBuffer[19].subindex 			:= 16#1A;
			eplReadBuffer[19].pData				:= ADR(readData.SLP);

			eplReadBuffer[20].name  	 		:= 'UFR'; //UNSIGNED
			eplReadBuffer[20].index 	 		:= 16#2042;
			eplReadBuffer[20].subindex 			:= 16#18;
			eplReadBuffer[20].pData				:= ADR(readData.UFR);

			eplReadBuffer[21].name  	 		:= 'BOA'; //Boost Enum, 0 Boost inactive, 1 boost dynamic, 2 boost static
			eplReadBuffer[21].index 	 		:= 16#206D;
			eplReadBuffer[21].subindex 			:= 16#B;
			eplReadBuffer[21].pData				:= ADR(readData.BOA);

			eplReadBuffer[22].name  	 		:= 'FAB'; //UNSIGNED
			eplReadBuffer[22].index 	 		:= 16#206D;
			eplReadBuffer[22].subindex 			:= 16#0C;
			eplReadBuffer[22].pData				:= ADR(readData.FAB);

			eplReadBuffer[23].name  	 		:= 'BOO'; //SIGNED
			eplReadBuffer[23].index 	 		:= 16#206D;
			eplReadBuffer[23].subindex 			:= 16#D;
			eplReadBuffer[23].pData				:= ADR(readData.BOO);

			//For Quadratic V/f
			eplReadBuffer[24].name  	 		:= 'PFL'; //UNSIGNED
			eplReadBuffer[24].index 	 		:= 16#2042;
			eplReadBuffer[24].subindex			:= 16#19;
			eplReadBuffer[24].pData				:= ADR(readData.PFL);

			//For 5pts mode
			eplReadBuffer[25].name  	 		:= 'F1'; //UNSIGNED
			eplReadBuffer[25].index 	 		:= 16#205E;
			eplReadBuffer[25].subindex 			:= 16#05;
			eplReadBuffer[25].pData				:= ADR(readData.F1);

			eplReadBuffer[26].name  	 		:= 'U1'; //UNSIGNED
			eplReadBuffer[26].index 	 		:= 16#205E;
			eplReadBuffer[26].subindex 			:= 16#04;
			eplReadBuffer[26].pData				:= ADR(readData.U1);

			eplReadBuffer[27].name  			:= 'F2'; //UNSIGNED
			eplReadBuffer[27].index 	 		:= 16#205E;
			eplReadBuffer[27].subindex 			:= 16#7;
			eplReadBuffer[27].pData				:= ADR(readData.F2);

			eplReadBuffer[28].name  	 		:= 'U2'; //UNSIGNED
			eplReadBuffer[28].index 	 		:= 16#205E;
			eplReadBuffer[28].subindex 			:= 16#6;
			eplReadBuffer[28].pData				:= ADR(readData.U2);

			eplReadBuffer[29].name  	 		:= 'F3'; //UNSIGNED
			eplReadBuffer[29].index	 			:= 16#205E;
			eplReadBuffer[29].subindex 			:= 16#09;
			eplReadBuffer[29].pData				:= ADR(readData.F3);

			eplReadBuffer[30].name  	 		:= 'U3'; //UNSIGNED
			eplReadBuffer[30].index 	 		:= 16#205E;
			eplReadBuffer[30].subindex 			:= 16#08;
			eplReadBuffer[30].pData				:= ADR(readData.U3);

			eplReadBuffer[31].name  	 		:= 'F4'; //UNSIGNED
			eplReadBuffer[31].index 	 		:= 16#205E;
			eplReadBuffer[31].subindex 			:= 16#0B;
			eplReadBuffer[31].pData				:= ADR(readData.F4);

			eplReadBuffer[32].name  	 		:= 'U4'; //UNSIGNED
			eplReadBuffer[32].index 	 		:= 16#205E;
			eplReadBuffer[32].subindex 			:= 16#0A;
			eplReadBuffer[32].pData				:= ADR(readData.U4);

			eplReadBuffer[33].name  	 		:= 'F5'; //UNSIGNED
			eplReadBuffer[33].index 	 		:= 16#205E;
			eplReadBuffer[33].subindex 			:= 16#D;
			eplReadBuffer[33].pData				:= ADR(readData.F5);

			eplReadBuffer[34].name  	 		:= 'U5'; //UNSIGNED
			eplReadBuffer[34].index 	 		:= 16#205E;
			eplReadBuffer[34].subindex 			:= 16#C;
			eplReadBuffer[34].pData				:= ADR(readData.U5);

			//End 5pts mode params

			//For vector control
			eplReadBuffer[35].name  	 		:= 'SIT'; //UNSIGNED
			eplReadBuffer[35].index 	 		:= 16#203D;
			eplReadBuffer[35].subindex 			:= 16#05;
			eplReadBuffer[35].pData				:= ADR(readData.SIT);

			eplReadBuffer[36].name  	 		:= 'SFC'; //UNSIGNED
			eplReadBuffer[36].index 	 		:= 16#203D;
			eplReadBuffer[36].subindex 			:= 16#06;
			eplReadBuffer[36].pData				:= ADR(readData.SFC);
			// End for vec control

			//Hysteresis & skip freq.
			eplReadBuffer[37].name  	 		:= ' JFH'; //UNSIGNED
			eplReadBuffer[37].index 	 		:= 16#2053;
			eplReadBuffer[37].subindex 			:= 16#0C;
			eplReadBuffer[37].pData				:= ADR(readData.JFH);

			eplReadBuffer[38].name  	 		:= 'JPF'; //UNSIGNED
			eplReadBuffer[38].index 	 		:= 16#2053;
			eplReadBuffer[38].subindex 			:= 16#02;
			eplReadBuffer[38].pData				:= ADR(readData.JPF);

			eplReadBuffer[39].name  	 		:= 'JF2'; //UNSIGNED
			eplReadBuffer[39].index 	 		:= 16#2053;
			eplReadBuffer[39].subindex 			:= 16#03;
			eplReadBuffer[39].pData				:= ADR(readData.JF2);

			eplReadBuffer[40].name  	 		:= 'JF3'; //UNSIGNED
			eplReadBuffer[40].index 	 		:= 16#2053;
			eplReadBuffer[40].subindex 			:= 16#04;
			eplReadBuffer[40].pData				:= ADR(readData.JF3);
			//End hyst. & skip freq.

			//Acceleration values
			eplReadBuffer[41].name  	 		:= 'SPA'; //UNSIGNED
			eplReadBuffer[41].index 	 		:= 16#2038;
			eplReadBuffer[41].subindex 			:= 16#0C;
			eplReadBuffer[41].pData				:= ADR(readData.SPA);

			eplReadBuffer[42].name  	 		:= 'SPAT'; //UNSIGNED
			eplReadBuffer[42].index 	 		:= 16#2038;
			eplReadBuffer[42].subindex 			:= 16#03;
			eplReadBuffer[42].pData				:= ADR(readData.SPAT);

			eplReadBuffer[43].name  	 		:= 'SPD'; //UNSIGNED
			eplReadBuffer[43].index 	 		:= 16#2038;
			eplReadBuffer[43].subindex 			:= 16#0F;
			eplReadBuffer[43].pData				:= ADR(readData.SPD);

			eplReadBuffer[44].name  	 		:= 'SPDT'; //UNSIGNED
			eplReadBuffer[44].index 	 		:= 16#2038;
			eplReadBuffer[44].subindex 			:= 16#11;
			eplReadBuffer[44].pData				:= ADR(readData.SPDT);

			eplReadBuffer[45].name  	 		:= 'RPT'; //Enum - Linear Ramp (0), S-ramp (1), U-Ramp (2), Customized (3)
			eplReadBuffer[45].index 	 		:= 16#203C;
			eplReadBuffer[45].subindex 			:= 16#05;
			eplReadBuffer[45].pData				:= ADR(readData.RPT);
			//End accel values

			//DC injection braking
			eplReadBuffer[46].name  	 		:= 'ADC'; //Enum - No DC inject(0), Yes (1), Continuous DC inj brake (2)
			eplReadBuffer[46].index 	 		:= 16#204A;
			eplReadBuffer[46].subindex 			:= 16#02;
			eplReadBuffer[46].pData				:= ADR(readData.ADC);

			eplReadBuffer[47].name  	 		:= 'FLR'; //Enum - catch spinning loads No(0), yes(1)
			eplReadBuffer[47].index 	 		:= 16#2001;
			eplReadBuffer[47].subindex 			:= 16#0B;
			eplReadBuffer[47].pData				:= ADR(readData.FLR);

			eplReadBuffer[48].name  	 		:= 'SDC1'; //UNSIGNED
			eplReadBuffer[48].index 	 		:= 16#204A;
			eplReadBuffer[48].subindex 			:= 16#04;
			eplReadBuffer[48].pData				:= ADR(readData.SDC1);

			eplReadBuffer[49].name  	 		:= 'TDC1'; //UNSIGNED
			eplReadBuffer[49].index 	 		:= 16#204A;
			eplReadBuffer[49].subindex 			:= 16#03;
			eplReadBuffer[49].pData				:= ADR(readData.TDC1);

			eplReadBuffer[50].name  	 		:= 'SDC2'; //UNSIGNED
			eplReadBuffer[50].index 	 		:= 16#204A;
			eplReadBuffer[50].subindex 			:= 16#06;
			eplReadBuffer[50].pData				:= ADR(readData.SDC2);

			eplReadBuffer[51].name  	 		:= 'TDC2'; //UNSIGNED
			eplReadBuffer[51].index 	 		:= 16#204A;
			eplReadBuffer[51].subindex 			:= 16#05;
			eplReadBuffer[51].pData				:= ADR(readData.TDC2);

			eplReadBuffer[52].name  	 		:= 'BRA'; //Enum - Braking cmd transistor(No) (0), Dec ramp adapt assinged (YES) (1), Dynamic high torque (2)
			eplReadBuffer[52].index 	 		:= 16#203C;
			eplReadBuffer[52].subindex 			:= 16#04;
			eplReadBuffer[52].pData				:= ADR(readData.BRA);

			eplReadBuffer[53].name  	 		:= 'DCF'; //UNSIGNED
			eplReadBuffer[53].index 	 		:= 16#2052;
			eplReadBuffer[53].subindex 			:= 16#1F;
			eplReadBuffer[53].pData				:= ADR(readData.DCF);

			eplReadBuffer[54].name  	 		:= 'IDC'; //UNSIGNED
			eplReadBuffer[54].index 	 		:= 16#2052;
			eplReadBuffer[54].subindex 			:= 16#0B;
			eplReadBuffer[54].pData				:= ADR(readData.IDC);

			eplReadBuffer[55].name  	 		:= 'TDI'; //UNSIGNED
			eplReadBuffer[55].index 	 		:= 16#2052;
			eplReadBuffer[55].subindex 			:= 16#0E;
			eplReadBuffer[55].pData				:= ADR(readData.TDI);

			eplReadBuffer[56].name  	 		:= 'IDC2'; //UNSIGNED
			eplReadBuffer[56].index 	 		:= 16#2052;
			eplReadBuffer[56].subindex 			:= 16#0D;
			eplReadBuffer[56].pData				:= ADR(readData.IDC2);

			eplReadBuffer[57].name  	 		:= 'TDC'; //UNSIGNED
			eplReadBuffer[57].index 	 		:= 16#2052;
			eplReadBuffer[57].subindex 			:= 16#0C;
			eplReadBuffer[57].pData				:= ADR(readData.TDC);

			//Load management
			eplReadBuffer[58].name  	 		:= 'ULT';	//UNSIGNED
			eplReadBuffer[58].index 	 		:= 16#2072;
			eplReadBuffer[58].subindex 			:= 16#0C;
			eplReadBuffer[58].pData				:= ADR(readData.ULT);

			eplReadBuffer[59].name  	 		:= 'LUL';  //UNSIGNED
			eplReadBuffer[59].index 	 		:= 16#2072;
			eplReadBuffer[59].subindex 			:= 16#10;
			eplReadBuffer[59].pData				:= ADR(readData.LUL);

			eplReadBuffer[60].name  	 		:= 'RMUD';
			eplReadBuffer[60].index 	 		:= 16#2072;
			eplReadBuffer[60].subindex 			:= 16#0F;
			eplReadBuffer[60].pData				:= ADR(readData.RMUD);

			eplReadBuffer[61].name  	 		:= 'LUN';
			eplReadBuffer[61].index 	 		:= 16#2072;
			eplReadBuffer[61].subindex 			:= 16#11;
			eplReadBuffer[61].pData				:= ADR(readData.LUN);

			eplReadBuffer[62].name  	 		:= 'FTU';
			eplReadBuffer[62].index 	 		:= 16#2072;
			eplReadBuffer[62].subindex 			:= 16#0E;
			eplReadBuffer[62].pData				:= ADR(readData.FTU);

			eplReadBuffer[63].name  	 		:= 'TOL';
			eplReadBuffer[63].index 	 		:= 16#2072;
			eplReadBuffer[63].subindex 			:= 16#16;
			eplReadBuffer[63].pData				:= ADR(readData.U3);

			eplReadBuffer[64].name  	 		:= 'LOC'; //UNSIGNED
			eplReadBuffer[64].index 	 		:= 16#2072;
			eplReadBuffer[64].subindex 			:= 16#1A;
			eplReadBuffer[64].pData				:= ADR(readData.LOC);

			eplReadBuffer[65].name  	 		:= 'FTO'; //UNSIGNED
			eplReadBuffer[65].index 			:= 16#2072;
			eplReadBuffer[65].subindex 			:= 16#18;
			eplReadBuffer[65].pData				:= ADR(readData.FTO);
			//end load management

			//Thermals

			eplReadBuffer[66].name  	 		:= 'ITH'; //UNSIGNED
			eplReadBuffer[66].index 	 		:= 16#2042;
			eplReadBuffer[66].subindex 			:= 16#17;
			eplReadBuffer[66].pData				:= ADR(readData.ITH);

			eplReadBuffer[67].name  	 		:= 'I2TA'; //Enumeration - 0 (no), 1 (yes)
			eplReadBuffer[67].index 	 		:= 16#2042;
			eplReadBuffer[67].subindex 			:= 16#20;
			eplReadBuffer[67].pData				:= ADR(readData.I2TA);
			//end thermals

			//Mains voltage monitoring

			eplReadBuffer[68].name  	 		:= 'MAINS'; //UNSIGNED 0.0V..6553.5V
			eplReadBuffer[68].index 	 		:= 16#2002;
			eplReadBuffer[68].subindex 			:= 16#08;
			eplReadBuffer[68].pData				:= ADR(readData.MAINS);

			startupstate := COPY;

			//Additional monitoring

			eplReadBuffer[69].name  	 		:= 'OTR'; //Motor Torque % -3276.7% .. 3276.7%
			eplReadBuffer[69].index 	 		:= 16#2042;
			eplReadBuffer[69].subindex 			:= 16#20;
			eplReadBuffer[69].measurementUnit	:= Percent;
			eplReadBuffer[69].pData				:= ADR(readData.OTR);

			(* Synchronous Motor Parameters *)

			//Pole pairs

			eplReadBuffer[70].name  	 		:= 'AST'; //Enum - Braking cmd transistor(No) (0), Dec ramp adapt assinged (YES) (1), Dynamic high torque (2)
			eplReadBuffer[70].index 	 		:= 16#2042;
			eplReadBuffer[70].subindex 			:= 16#49;
			eplReadBuffer[70].measurementUnit	:= Undefined;
			eplReadBuffer[70].pData				:= ADR(readData.PPNS);

			//Sync speed

			eplReadBuffer[71].name  	 		:= 'NSPS'; //Synchronous nominal speed
			eplReadBuffer[71].index 	 		:= 16#2042;
			eplReadBuffer[71].subindex 			:= 16#48;
			eplReadBuffer[71].measurementUnit	:= RPM;
			eplReadBuffer[71].pData				:= ADR(readData.NSPS);

			//Sync speed

			eplReadBuffer[72].name  	 		:= 'NCRS'; //Synchronous nominal current
			eplReadBuffer[72].index 	 		:= 16#2042;
			eplReadBuffer[72].subindex 			:= 16#47;
			eplReadBuffer[72].measurementUnit	:= Amps;
			eplReadBuffer[72].pData				:= ADR(readData.NCRS);

			eplReadBuffer[73].name  	 		:= 'TQS'; //Synchronous motor torque
			eplReadBuffer[73].index 	 		:= 16#2042;
			eplReadBuffer[73].subindex 			:= 16#55;
			eplReadBuffer[73].measurementUnit	:= NewtonMeter;
			eplReadBuffer[73].pData				:= ADR(readData.TQS);

			eplReadBuffer[74].name  	 		:= 'RSAS'; //Synchronous motor stator resistance
			eplReadBuffer[74].index 	 		:= 16#2042;
			eplReadBuffer[74].subindex 			:= 16#53;
			eplReadBuffer[74].measurementUnit	:= Ohm;
			eplReadBuffer[74].pData				:= ADR(readData.RSAS);

			eplReadBuffer[75].name  	 		:= 'LDS'; //Synchronous motor stator resistance
			eplReadBuffer[75].index 	 		:= 16#2042;
			eplReadBuffer[75].subindex 			:= 16#4B;
			eplReadBuffer[75].measurementUnit	:= Millihenry;
			eplReadBuffer[75].pData				:= ADR(readData.LDS);

			eplReadBuffer[76].name  	 		:= 'LQS'; //Synchronous motor stator resistance
			eplReadBuffer[76].index 	 		:= 16#2042;
			eplReadBuffer[76].subindex 			:= 16#4C;
			eplReadBuffer[76].measurementUnit	:= Millihenry;
			eplReadBuffer[76].pData				:= ADR(readData.LQS);

			eplReadBuffer[77].name  	 		:= 'PHS'; //Synchronous motor stator resistance
			eplReadBuffer[77].index 	 		:= 16#2042;
			eplReadBuffer[77].subindex 			:= 16#4A;
			eplReadBuffer[77].measurementUnit	:= Undefined; 		// mV/rpm or V/1000rpm
			eplReadBuffer[77].pData				:= ADR(readData.PHS);

		COPY:
			//Assign the same addresses to the write buffer

			FOR i := 0  TO MAXINDEX DO
				eplWriteBuffer[i].name  		:= eplReadBuffer[i].name;
				eplWriteBuffer[i].index 		:= eplReadBuffer[i].index;
				eplWriteBuffer[i].subindex		:= eplReadBuffer[i].subindex;

				//Read and write all parameters by default
				readBools[i] := TRUE;
				writeBools[i] := TRUE;
			END_FOR

			//Assign links to writeBuffer

			eplWriteBuffer[0].pData				:= ADR(writeData.NSP);
			eplWriteBuffer[1].pData				:= ADR(writeData.FRS);
			eplWriteBuffer[2].pData				:= ADR(writeData.UNS);
			eplWriteBuffer[3].pData				:= ADR(writeData.NCR);
			eplWriteBuffer[4].pData				:= ADR(writeData.COSINE);
			eplWriteBuffer[5].pData				:= ADR(writeData.NPR);
			eplWriteBuffer[6].pData				:= ADR(writeData.TUN);
			eplWriteBuffer[7].pData				:= ADR(writeData.RSA);
			eplWriteBuffer[8].pData				:= ADR(writeData.LFA);
			eplWriteBuffer[9].pData				:= ADR(writeData.IDA);
			eplWriteBuffer[10].pData			:= ADR(writeData.TRA);
			eplWriteBuffer[11].pData			:= ADR(writeData.SFR);
			eplWriteBuffer[12].pData			:= ADR(writeData.SFT);
			eplWriteBuffer[13].pData			:= ADR(writeData.NRD);
			eplWriteBuffer[14].pData			:= ADR(writeData.CTT);
			eplWriteBuffer[15].pData			:= ADR(writeData.SPGU);
			eplWriteBuffer[16].pData			:= ADR(writeData.SPG);
			eplWriteBuffer[17].pData			:= ADR(writeData.FFH);
			eplWriteBuffer[18].pData			:= ADR(writeData.CRTF);
			eplWriteBuffer[19].pData			:= ADR(writeData.SLP);
			eplWriteBuffer[20].pData			:= ADR(writeData.UFR);
			eplWriteBuffer[21].pData			:= ADR(writeData.BOA);
			eplWriteBuffer[22].pData			:= ADR(writeData.FAB);
			eplWriteBuffer[23].pData			:= ADR(writeData.BOO);
			eplWriteBuffer[24].pData			:= ADR(writeData.PFL);
			eplWriteBuffer[25].pData			:= ADR(writeData.F1);
			eplWriteBuffer[26].pData			:= ADR(writeData.U1);
			eplWriteBuffer[27].pData			:= ADR(writeData.F2);
			eplWriteBuffer[28].pData			:= ADR(writeData.U2);
			eplWriteBuffer[29].pData			:= ADR(writeData.F3);
			eplWriteBuffer[30].pData			:= ADR(writeData.U3);
			eplWriteBuffer[31].pData			:= ADR(writeData.F4);
			eplWriteBuffer[32].pData			:= ADR(writeData.U4);
			eplWriteBuffer[33].pData			:= ADR(writeData.F5);
			eplWriteBuffer[34].pData			:= ADR(writeData.U5);
			eplWriteBuffer[35].pData			:= ADR(writeData.SIT);
			eplWriteBuffer[36].pData			:= ADR(writeData.SFC);
			eplWriteBuffer[37].pData			:= ADR(writeData.JFH);
			eplWriteBuffer[38].pData			:= ADR(writeData.JPF);
			eplWriteBuffer[39].pData			:= ADR(writeData.JF2);
			eplWriteBuffer[40].pData			:= ADR(writeData.JF3);
			eplWriteBuffer[41].pData			:= ADR(writeData.SPA);
			eplWriteBuffer[42].pData			:= ADR(writeData.SPAT);
			eplWriteBuffer[43].pData			:= ADR(writeData.SPD);
			eplWriteBuffer[44].pData			:= ADR(writeData.SPDT);
			eplWriteBuffer[45].pData			:= ADR(writeData.RPT);
			eplWriteBuffer[46].pData			:= ADR(writeData.ADC);
			eplWriteBuffer[47].pData			:= ADR(writeData.FLR);
			eplWriteBuffer[48].pData			:= ADR(writeData.SDC1);
			eplWriteBuffer[49].pData			:= ADR(writeData.TDC1);
			eplWriteBuffer[50].pData			:= ADR(writeData.SDC2);
			eplWriteBuffer[51].pData			:= ADR(writeData.TDC2);
			eplWriteBuffer[52].pData			:= ADR(writeData.BRA);
			eplWriteBuffer[53].pData			:= ADR(writeData.DCF);
			eplWriteBuffer[54].pData			:= ADR(writeData.IDC);
			eplWriteBuffer[55].pData			:= ADR(writeData.TDI);
			eplWriteBuffer[56].pData			:= ADR(writeData.IDC2);
			eplWriteBuffer[57].pData			:= ADR(writeData.TDC);
			eplWriteBuffer[58].pData			:= ADR(writeData.ULT);
			eplWriteBuffer[59].pData			:= ADR(writeData.LUL);
			eplWriteBuffer[60].pData			:= ADR(writeData.RMUD);
			eplWriteBuffer[61].pData			:= ADR(writeData.LUN);
			eplWriteBuffer[61].pData			:= ADR(writeData.FTU);
			eplWriteBuffer[63].pData			:= ADR(writeData.TOL);
			eplWriteBuffer[64].pData			:= ADR(writeData.LOC);
			eplWriteBuffer[65].pData			:= ADR(writeData.FTO);
			eplWriteBuffer[66].pData			:= ADR(writeData.ITH);
			eplWriteBuffer[67].pData			:= ADR(writeData.I2TA);
			eplWriteBuffer[68].pData			:= ADR(writeData.OTR);
			eplWriteBuffer[69].pData			:= ADR(writeData.MAINS);
			eplWriteBuffer[70].pData			:= ADR(writeData.PPNS);
			eplWriteBuffer[71].pData			:= ADR(writeData.NSPS);
			eplWriteBuffer[72].pData			:= ADR(writeData.NCRS);
			eplWriteBuffer[73].pData			:= ADR(writeData.TQS);
			eplWriteBuffer[74].pData			:= ADR(writeData.RSAS);
			eplWriteBuffer[75].pData			:= ADR(writeData.LDS);
			eplWriteBuffer[76].pData			:= ADR(writeData.LQS);
			eplWriteBuffer[77].pData			:= ADR(writeData.PHS);

			i := 0;
			startupstate := FIRSTREAD;

		FIRSTREAD:

		eplReadBlock.enable 	:= TRUE;
		eplReadBlock.index 		:= eplReadBuffer[i].index;
		eplReadBlock.subindex 	:= eplReadBuffer[i].subindex;
		eplReadBlock.node  		:= hmiCom.NodeNumber;
		eplReadBlock.pData 		:= eplReadBuffer[i].pData;
		eplReadBlock.datalen 	:= SIZEOF(readData.ADC);	//Any will do since the max is 2 bytes

		IF eplReadBlock.status = 0 THEN
			eplReadBlock.enable := 0;
			i := i + 1;
		END_IF

		IF i = MAXINDEX THEN
			eplReadBlock.enable := FALSE;
			hmiCom.ReadWriteBuffer := readData;
			startupstate := DONE;
		END_IF

		eplReadBlock();

		DONE:

			startupDone := TRUE;

	END_CASE

END_ACTION
```

- Visualisation Logical/mappView (not shown)

Listed in the project but not available here: Logical/Global.typ, Logical/Global.var
